FUNCTION Convert_DT_TO_DT : BOOL
VAR_INPUT
	in : DT;
	out : REFERENCE TO DT;
END_VAR

out := in;
Convert_DT_TO_DT := TRUE;

END_FUNCTION

(* stored: Version 1.1.0.1, ProductVersion 3.1.4024.12
   POU Convert_DT_TO_DT: Id {c252d7fe-e597-48d5-9bcd-6abb433f9cb9}, SpecialFunc None *)
